TYPE ST_CSL_Hmi :
STRUCT
	Home_page		: BOOL;
	Allarms_page	: BOOL;
	Numbers_page	: BOOL;
END_STRUCT
END_TYPE

(* stored: Version 1.1.0.1, ProductVersion 3.1.4024.12
   DUT ST_CSL_Hmi: Id {f7a7f018-6f3d-404c-8f7e-da5ba158cdd1} *)
